Universal Robots PolyScope program: Socket_klep_test1.urp

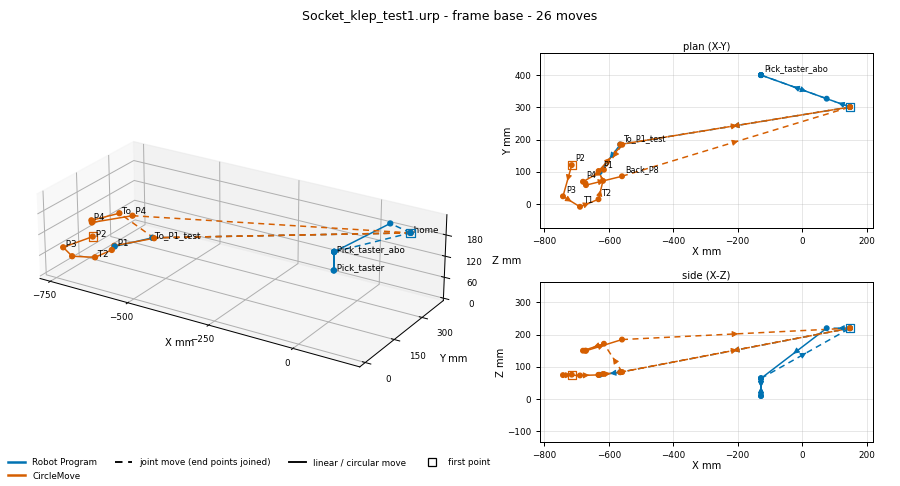
[picture p0: tool path of Socket_klep_test1.urp in frame base, 26 of 27 moves have a stored position in this frame; points joined in program order, loops and branches not executed]
Program Socket_klep_test1 (createdIn=3.0.16471.0 lastSavedIn=3.3.4.310 directory=/programs/PPAU/ITIS installation=Fomeco_1 robotSerialNumber=2014300380)
Calibrated DH parameters: a=[0.000017, -0.607894, -0.567863, -0.000043, 0.000045, 0]; d=[0.128178, 49.570862, -69.933448, 20.52608, 0.115764, 0.091962]; alpha=[1.571183, -0.001568, -0.003173, 1.570373, -1.570911, 0]; deltaTheta=[-0.000009, -0.127231, 0.240463, -0.113236, -0.000061, 0.000049]
BeforeStart
  socket_ip := "10.32.3.54"
  SuppressedNode
    socket_ip := "192.168.2.14"
  socket_port := 30000
  socket_name := "test"
  request_pose := "request_pose"
  request_leaks := "request_leaks"
  eof := False
  SuppressedNode
    URCap com.robotiq.urcap.gripper.GripperNode data=position = 100
      | force = 0
      | speed = 100
      | blocking = true
  recording := False
  Taster_Picked := 0
  Drop_off := 0
Robot Program (runOnlyOnce=true motionType=MoveJ speed=1.047198 acceleration=1.396263 recalculateMotions=false)
  var_1 := socket_open(socket_ip,socket_port, socket_name)
  MoveJ speed 60 deg/s, acceleration 80 deg/s^2 (recalculateMotions=false)
    Waypoint home: TCP in base x=148.583 y=300.967 z=219.982 mm, rx=0.029 ry=-1.5747 rz=0.0389 rad; joints [65.958, -63.946, -124.118, -82.153, 89.459, -206.464] deg; flange x=317.193 y=310.053 z=505.621 mm, rx=-0.0678 ry=3.1367 rz=-0.0099 rad
  Loop While (checkContinuously=false) expression=var_1≟ False
    var_1 := socket_open(socket_ip,socket_port, socket_name)
    Wait Sleep waitTime=0.5
  MoveJ speed 60 deg/s, acceleration 80 deg/s^2 (recalculateMotions=false)
    Waypoint socket_OK: TCP in base x=76.144 y=326.862 z=219.973 mm, rx=0.2097 ry=-1.5649 rz=0.2189 rad; joints [79.114, -63.946, -124.118, -82.153, 89.459, -206.464] deg; flange x=238.303 y=374.107 z=505.621 mm, rx=-0.4265 ry=3.1076 rz=-0.0091 rad
  Popup Message (haltProgram=false message=Is the needle into the gripper? Taster_Picked=1?)
  SuppressedNode
    Loop While (checkContinuously=false) expression=var_1≟ False
      var_1 := socket_open(socket_ip, socket_port, socket_name)
      Wait Sleep waitTime=0.5
  If Taster_Picked≟0
    SuppressedNode
      URCap com.robotiq.urcap.gripper.GripperNode data=position = 0
        | force = 0
        | speed = 100
        | blocking = true
    URCap com.robotiq.urcap.gripper.GripperNode data=position = 39
      | force = 0
      | speed = 100
      | blocking = true
    SuppressedNode
      MoveJ speed 60 deg/s, acceleration 80 deg/s^2 (recalculateMotions=false)
        Waypoint Tussenp_1: motionParameters(blendRadius=0.05); TCP in base x=407.573 y=31.262 z=426.428 mm, rx=-2.2099 ry=-2.2302 rz=0.0042 rad; joints [27.849, -61.448, -133.482, -75.247, 89.892, -152.644] deg
    MoveL speed 250 mm/s, acceleration 1200 mm/s^2 (recalculateMotions=false) feature=Base
      Waypoint Pick_taster_abo: TCP in base x=-127.718 y=400.102 z=64.182 mm, rx=-0.0011 ry=-1.57 rz=0.0015 rad; joints [107.791, -64.197, -140.438, -65.442, 89.909, -162.223] deg; flange x=42.465 y=400.626 z=349.043 mm, rx=0.0004 ry=-3.1408 rz=0.0028 rad
      Waypoint Pick_taster: TCP in base x=-127.724 y=400.033 z=9.767 mm, rx=-0.0012 ry=-1.5701 rz=0.0017 rad; joints [107.802, -68.219, -144.624, -57.235, 89.914, -162.232] deg; flange x=42.468 y=400.612 z=294.675 mm, rx=0.0004 ry=-3.1408 rz=0.0028 rad
      SuppressedNode
        URCap com.robotiq.urcap.gripper.GripperNode data=position = 100
          | force = 0
          | speed = 0
          | blocking = true
      URCap com.robotiq.urcap.gripper.GripperNode data=position = 56
        | force = 100
        | speed = 100
        | blocking = true
      Waypoint Pick_taster_abo: TCP in base x=-127.718 y=400.102 z=64.182 mm, rx=-0.0011 ry=-1.57 rz=0.0015 rad; joints [107.791, -64.197, -140.438, -65.442, 89.909, -162.223] deg; flange x=42.465 y=400.626 z=349.043 mm, rx=0.0004 ry=-3.1408 rz=0.0028 rad
    Taster_Picked := 1
  Else 
    If Drop_off≟1
      SuppressedNode
        MoveJ speed 60 deg/s, acceleration 80 deg/s^2 (recalculateMotions=false)
          Waypoint Tussenp_1: motionParameters(blendRadius=0.05); TCP in base x=407.573 y=31.262 z=426.428 mm, rx=-2.2099 ry=-2.2302 rz=0.0042 rad; joints [27.849, -61.448, -133.482, -75.247, 89.892, -152.644] deg
      MoveL speed 250 mm/s, acceleration 1200 mm/s^2 (recalculateMotions=false) feature=Base
        Waypoint Pick_taster_abo: TCP in base x=-127.718 y=400.102 z=64.182 mm, rx=-0.0011 ry=-1.57 rz=0.0015 rad; joints [107.791, -64.197, -140.438, -65.442, 89.909, -162.223] deg; flange x=42.465 y=400.626 z=349.043 mm, rx=0.0004 ry=-3.1408 rz=0.0028 rad
        Waypoint Pick_taster: TCP in base x=-127.724 y=400.033 z=9.767 mm, rx=-0.0012 ry=-1.5701 rz=0.0017 rad; joints [107.802, -68.219, -144.624, -57.235, 89.914, -162.232] deg; flange x=42.468 y=400.612 z=294.675 mm, rx=0.0004 ry=-3.1408 rz=0.0028 rad
        URCap com.robotiq.urcap.gripper.GripperNode data=position = 39
          | force = 0
          | speed = 100
          | blocking = true
        Waypoint Pick_taster_abo: TCP in base x=-127.718 y=400.102 z=64.182 mm, rx=-0.0011 ry=-1.57 rz=0.0015 rad; joints [107.791, -64.197, -140.438, -65.442, 89.909, -162.223] deg; flange x=42.465 y=400.626 z=349.043 mm, rx=0.0004 ry=-3.1408 rz=0.0028 rad
      SuppressedNode
        MoveJ speed 60 deg/s, acceleration 80 deg/s^2 (recalculateMotions=false)
          Waypoint Tussenp_1: motionParameters(blendRadius=0.05); TCP in base x=407.573 y=31.262 z=426.428 mm, rx=-2.2099 ry=-2.2302 rz=0.0042 rad; joints [27.849, -61.448, -133.482, -75.247, 89.892, -152.644] deg
      MoveJ speed 60 deg/s, acceleration 80 deg/s^2 (recalculateMotions=false)
        Waypoint Home: TCP in base x=148.6 y=300.933 z=219.943 mm, rx=0.029 ry=-1.5747 rz=0.039 rad; joints [65.958, -63.946, -124.118, -82.153, 89.459, -206.464] deg; flange x=317.193 y=310.053 z=505.621 mm, rx=-0.0678 ry=3.1367 rz=-0.0099 rad
      Halt
  MoveJ speed 60 deg/s, acceleration 80 deg/s^2 (recalculateMotions=false)
    SuppressedNode
      Waypoint To_P1: TCP in base x=-557.811 y=178.532 z=83.365 mm, rx=0.662 ry=-1.4749 rz=0.6549 rad; joints [163.403, -80.044, -128.08, -61.958, 89.394, -154.861] deg; flange x=-445.689 y=303.494 z=369.672 mm, rx=-1.2818 ry=2.8616 rz=0.0072 rad
    Waypoint To_P1_test: TCP in base x=-564.523 y=184.862 z=83.39 mm, rx=0.6205 ry=-1.4875 rz=0.6129 rad; joints [163.403, -80.044, -128.08, -61.958, 89.394, 208.234] deg; flange x=-445.689 y=303.494 z=369.672 mm, rx=-1.2041 ry=2.8953 rz=0.0074 rad
  recording := True
  MoveP speed 20 mm/s, acceleration 80 mm/s^2 (blendRadius=0.001 recalculateMotions=false) feature=Base
    Waypoint P1: TCP in base x=-628.014 y=99.393 z=75.306 mm, rx=0.58 ry=-1.4987 rz=0.5721 rad; joints [174.614, -81.228, -128.051, -60.883, 89.421, 222.44] deg; flange x=-502.991 y=211.646 z=361.466 mm, rx=-1.1281 ry=2.926 rz=0.0076 rad
    SuppressedNode
      Call send_pos_leak
    CircleMove
      Waypoint P2: TCP in base x=-714.974 y=120.772 z=75.776 mm, rx=1.73 ry=-0.7731 rz=1.7309 rad; joints [174.452, -110.913, -94.631, -64.612, 89.374, 132.204] deg; flange x=-830.236 y=244.791 z=361.184 mm, rx=-2.8659 ry=1.2688 rz=-0.0008 rad
      Waypoint P3: TCP in base x=-742.257 y=23.865 z=74.391 mm, rx=-1.8242 ry=-0.6373 rz=-1.8353 rad; joints [196.193, -112.289, -92.949, -65.063, 89.45, 67.503] deg; flange x=-875.984 y=-84.385 z=358.212 mm, rx=-2.9594 ry=-1.0388 rz=-0.0089 rad
    CircleMove
      Waypoint T1: TCP in base x=-689.438 y=-8.604 z=73.377 mm, rx=-1.2305 ry=-1.1885 rz=-1.243 rad; joints [207.614, -98.432, -111.343, -60.576, 89.543, 29.784] deg; flange x=-696.964 y=-180.44 z=357.232 mm, rx=-2.2616 ry=-2.1771 rz=-0.0113 rad
      Waypoint T2: TCP in base x=-631.992 y=14.732 z=75.025 mm, rx=-0.6756 ry=-1.4616 rz=-0.6881 rad; joints [210.347, -80.397, -128.892, -61.082, 89.593, -9.634] deg; flange x=-523.864 y=-117.548 z=359.538 mm, rx=1.3281 ry=2.8465 rz=0.012 rad
    CircleMove
      Waypoint T3: TCP in base x=-618.088 y=71.772 z=77.887 mm, rx=-0.0141 ry=-1.5743 rz=-0.0248 rad; joints [192.794, -70.307, -135.479, -64.5, 89.501, -75.787] deg; flange x=-449.187 y=65.6 z=363.476 mm, rx=0.0388 ry=3.1377 rz=0.0106 rad
      Waypoint T4: TCP in base x=-631.644 y=102.42 z=75.309 mm, rx=0.6606 ry=-1.4758 rz=0.6531 rad; joints [173.148, -83.462, -126.161, -60.544, 89.401, -144.992] deg; flange x=-519.239 y=227.08 z=361.642 mm, rx=-1.2785 ry=2.8628 rz=0.0072 rad
    SuppressedNode
      Call send_pos_leak
    Waypoint Back1: TCP in base x=-558.414 y=183.88 z=83.894 mm, rx=0.6604 ry=-1.4757 rz=0.6532 rad; joints [162.876, -80.369, -127.76, -61.963, 89.383, -155.259] deg; flange x=-446.107 y=308.591 z=370.194 mm, rx=-1.2785 ry=2.8628 rz=0.0071 rad
  MoveJ speed 50 deg/s, acceleration 70 deg/s^2 (recalculateMotions=false)
    Waypoint To_P4: TCP in base x=-615.17 y=106.275 z=171.769 mm, rx=0.3917 ry=-1.8325 rz=0.4264 rad; joints [179.548, -81.89, -110.385, -94.458, 86.672, -118.783] deg; flange x=-555.326 y=172.063 z=491.487 mm, rx=-0.7098 ry=2.7551 rz=-0.0301 rad
  MoveP speed 10 mm/s, acceleration 50 mm/s^2 (blendRadius=0.001 recalculateMotions=false) feature=Base
    Waypoint P4: TCP in base x=-680.107 y=69.217 z=150.178 mm, rx=0.3918 ry=-1.8325 rz=0.4264 rad; joints [182.888, -87.801, -107.255, -91.824, 87.628, -115.588] deg; flange x=-620.279 y=135.045 z=469.893 mm, rx=-0.7098 ry=2.7551 rz=-0.0301 rad
    CircleMove
      Waypoint P5: TCP in base x=-672.687 y=64.573 z=150.309 mm, rx=0.3051 ry=-1.8485 rz=0.3087 rad; joints [185.186, -85.748, -108.982, -92.224, 88.296, -106.157] deg; flange x=-603.935 y=110.924 z=471.672 mm, rx=-0.5346 ry=2.7938 rz=-0.0031 rad
      Waypoint P6: TCP in base x=-670.877 y=58.582 z=149.91 mm, rx=0.2307 ry=-1.8576 rz=0.2078 rad; joints [187.441, -84.655, -109.935, -92.407, 88.955, -97.806] deg; flange x=-596.394 y=87.509 z=471.968 mm, rx=-0.3829 ry=2.8188 rz=0.0199 rad
    SuppressedNode
      CircleMove
        Waypoint P7: TCP in base x=-671.566 y=61.834 z=149.807 mm, rx=0.22 ry=-1.8586 rz=0.1936 rad; joints [187.371, -84.669, -109.921, -92.408, 88.936, -97.001] deg; flange x=-596.437 y=88.245 z=471.985 mm, rx=-0.3614 ry=2.8217 rz=0.0231 rad
        Waypoint P8: TCP in base x=-671.346 y=59.518 z=149.486 mm, rx=0.203 ry=-1.86 rz=0.1706 rad; joints [187.983, -84.473, -110.127, -92.406, 89.115, -94.991] deg; flange x=-595.195 y=81.886 z=471.673 mm, rx=-0.3263 ry=2.8262 rz=0.0284 rad
    Waypoint Back_P8: TCP in base x=-559.078 y=86.13 z=184.735 mm, rx=0.203 ry=-1.86 rz=0.1704 rad; joints [186.74, -72.671, -115.772, -98.546, 88.773, -96.168] deg; flange x=-482.956 y=108.419 z=506.947 mm, rx=-0.3263 ry=2.8262 rz=0.0284 rad
  recording := False
  Wait Sleep waitTime=1
  SuppressedNode
    Popup Message (haltProgram=false message=received?)
  MoveJ speed 60 deg/s, acceleration 80 deg/s^2 (recalculateMotions=false)
    Waypoint home: TCP in base x=148.583 y=300.967 z=219.982 mm, rx=0.029 ry=-1.5747 rz=0.0389 rad; joints [65.958, -63.946, -124.118, -82.153, 89.459, -206.464] deg; flange x=317.193 y=310.053 z=505.621 mm, rx=-0.0678 ry=3.1367 rz=-0.0099 rad
  Script: socket_send_string(request_leaks, socket_name)
  Wait Sleep waitTime=0.1
  s_str := socket_read_ascii_float(7, socket_name)
  nr_leaks := s_str[1]
  Popup Message (haltProgram=false message=ready to check leaks?)
  MoveJ speed 60 deg/s, acceleration 80 deg/s^2 (recalculateMotions=false)
    SuppressedNode
      Waypoint To_P1: TCP in base x=-557.811 y=178.532 z=83.365 mm, rx=0.662 ry=-1.4749 rz=0.6549 rad; joints [163.403, -80.044, -128.08, -61.958, 89.394, -154.861] deg; flange x=-445.689 y=303.494 z=369.672 mm, rx=-1.2818 ry=2.8616 rz=0.0072 rad
    Waypoint To_P1_test: TCP in base x=-564.523 y=184.862 z=83.39 mm, rx=0.6205 ry=-1.4875 rz=0.6129 rad; joints [163.403, -80.044, -128.08, -61.958, 89.394, 208.234] deg; flange x=-445.689 y=303.494 z=369.672 mm, rx=-1.2041 ry=2.8953 rz=0.0074 rad
  Loop While (checkContinuously=false) expression=eof≟ False
    Call get_pose
  SuppressedNode
    Loop While (checkContinuously=false) expression=s_str[0]≟0
      Placeholder
  Script: socket_close(socket_name="test")
  MoveJ speed 60 deg/s, acceleration 80 deg/s^2 (recalculateMotions=false)
    Waypoint home: TCP in base x=148.583 y=300.967 z=219.982 mm, rx=0.029 ry=-1.5747 rz=0.0389 rad; joints [65.958, -63.946, -124.118, -82.153, 89.459, -206.464] deg; flange x=317.193 y=310.053 z=505.621 mm, rx=-0.0678 ry=3.1367 rz=-0.0099 rad
SubProgram -> get_pose
SubProgram -> send_pos_leak
SubProgram send_pos_no_lea (keepSynchronizedWithDisk=false trackProgramExecution=false)
  SuppressedNode
    this_wp := get_actual_tcp_pose()
  this_wp := get_forward_kin()
  leak_flag := "no_leak"
  Script: socket_send_string(leak_flag, socket_name)
  Wait Sleep waitTime=0.02
  Script: socket_send_string(this_wp, socket_name)
Thread Thread_1 (runOnlyOnce=false trackProgramExecution=false)
  Loop Forever
    If digital_in[4]≟ True
      Call send_pos_leak
    btnState := digital_in[4]
    Wait Condition expression=btnState≠digital_in[4]
Thread Thread_2 (runOnlyOnce=false trackProgramExecution=false)
  Loop Forever
    Wait Sleep waitTime=0.25
    If recording≟ True
      Call send_pos_no_lea
SubProgram send_pos_leak (keepSynchronizedWithDisk=false trackProgramExecution=false)
  SuppressedNode
    this_wp := get_actual_tcp_pose()
  this_wp := get_forward_kin()
  leak_flag := "leak"
  Script: socket_send_string(leak_flag, socket_name)
  Script: socket_send_string(this_wp, socket_name)
SubProgram get_pose (keepSynchronizedWithDisk=false trackProgramExecution=false)
  Script: socket_send_string(request_pose, socket_name)
  s_str := socket_read_ascii_float(7, socket_name)
  var_3 := s_str[0]
  var_4 := s_str[1]
  If s_str[0]≟7
    this_wp := p[s_str[1], s_str[2], s_str[3], s_str[4], s_str[5], s_str[6]]
    SuppressedNode
      MoveJ speed 60 deg/s, acceleration 80 deg/s^2 (recalculateMotions=false)
        Waypoint Waypoint (Variable): variable=this_wp
    SuppressedNode
      var_2 := get_forward_kin()
    tool_offset := p[0,0,-0.01,0,0,0]
    this_wp := pose_trans(this_wp, tool_offset)
    MoveP speed 100 mm/s, acceleration 200 mm/s^2 (blendRadius=0.001 recalculateMotions=false) feature=Base
      Waypoint Waypoint (Variable): variable=this_wp
    SuppressedNode
      Wait Sleep waitTime=1
    If s_str[7]≟1
      Popup Message (haltProgram=false message=next leak?)
  If s_str[0]≟0
    Popup Message (haltProgram=false message=end of list)
    eof := True
